// TwinCAT 3 PLC project plcproject
// ProgramVersion: 3.1.4023.0
// libraries:
//   Tc2_Standard, * (Beckhoff Automation GmbH)
//   Tc2_System, * (Beckhoff Automation GmbH)
//   Tc3_Module, * (Beckhoff Automation GmbH)
// project tree:
//   DUTs/ POU2.TcPOU
//   / PlcTask.TcTTO
//   POUs/ MAIN.TcPOU
// real-time tasks:
//   TASK PlcTask: cycle T#10ms, priority 20, ADS port 350

CONFIGURATION plcproject
    RESOURCE PLC ON TwinCAT3
        TASK PlcTask(INTERVAL := T#10ms, PRIORITY := 20);
        PROGRAM MAIN WITH PlcTask : MAIN;
    END_RESOURCE
END_CONFIGURATION

// ---- POUs/MAIN.TcPOU
PROGRAM MAIN
VAR
	varprueba: BOOL;
	modifi: INT;
	apocoyes: INT;
	cambio2: INT;
	rndid: INT;
END_VAR

varprueba:= TRUE;

modifi:=2;


apocoyes:=3;


cambio2:=3;

rndid:=3;

END_PROGRAM

// ---- DUTs/POU2.TcPOU
PROGRAM POU2
VAR
	puvar2: INT;
END_VAR

puvar2:=4;

END_PROGRAM
